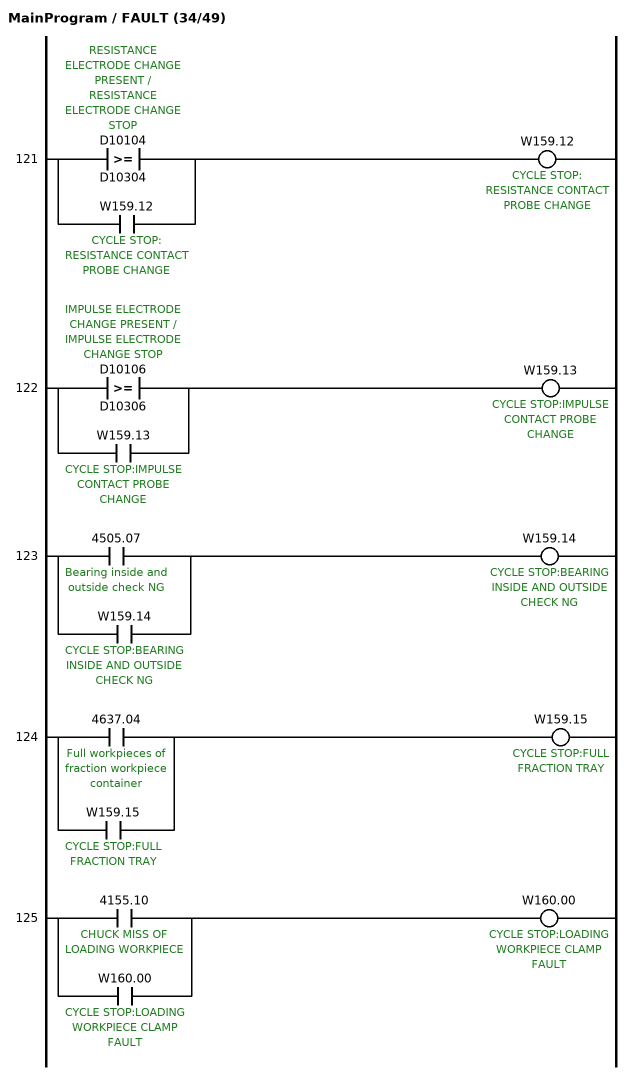
; [picture p96: MainProgram / FAULT, rungs 121-125]
; rung 121
LD>=L(326) D10104 D10304  ; RESISTANCE ELECTRODE CHANGE PRESENT, RESISTANCE ELECTRODE CHANGE STOP
OR W159.12  ; CYCLE STOP:RESISTANCE CONTACT PROBE CHANGE
OUT W159.12  ; CYCLE STOP:RESISTANCE CONTACT PROBE CHANGE
; rung 122
LD>=L(326) D10106 D10306  ; IMPULSE ELECTRODE CHANGE PRESENT, IMPULSE ELECTRODE CHANGE STOP
OR W159.13  ; CYCLE STOP:IMPULSE CONTACT PROBE CHANGE
OUT W159.13  ; CYCLE STOP:IMPULSE CONTACT PROBE CHANGE
; rung 123
LD 4505.07  ; Bearing inside and outside check NG
OR W159.14  ; CYCLE STOP:BEARING INSIDE AND OUTSIDE CHECK NG
OUT W159.14  ; CYCLE STOP:BEARING INSIDE AND OUTSIDE CHECK NG
; rung 124
LD 4637.04  ; Full workpieces of fraction workpiece container
OR W159.15  ; CYCLE STOP:FULL FRACTION TRAY
OUT W159.15  ; CYCLE STOP:FULL FRACTION TRAY
; rung 125
LD 4155.10  ; CHUCK MISS OF LOADING WORKPIECE
OR W160.00  ; CYCLE STOP:LOADING WORKPIECE CLAMP FAULT
OUT W160.00  ; CYCLE STOP:LOADING WORKPIECE CLAMP FAULT

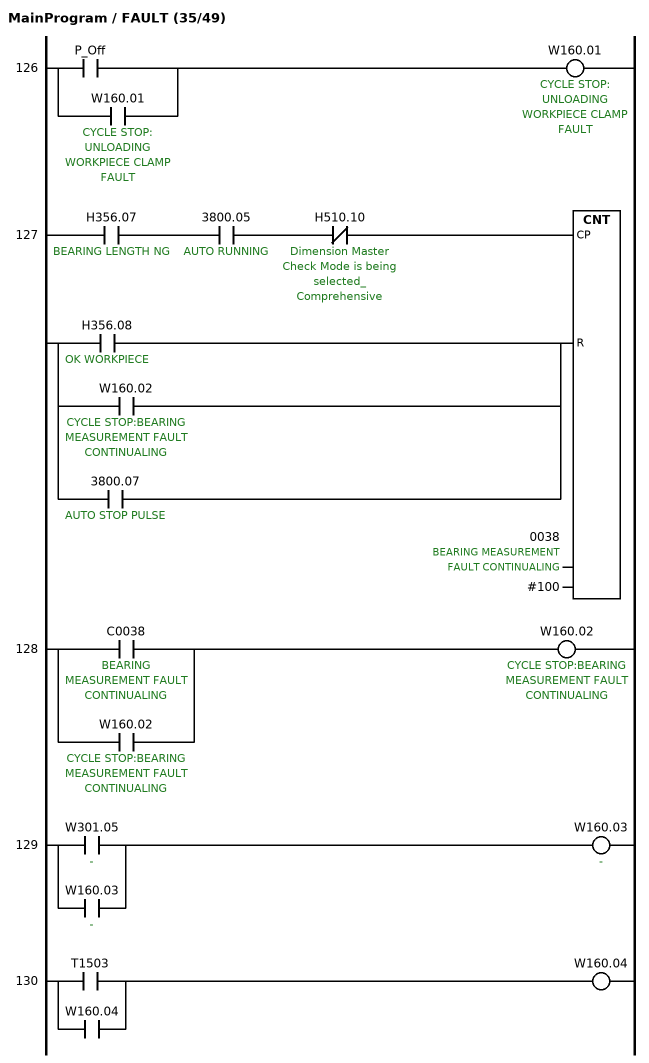
; rung 126
LD P_Off
OR W160.01  ; CYCLE STOP:UNLOADING WORKPIECE CLAMP FAULT
OUT W160.01  ; CYCLE STOP:UNLOADING WORKPIECE CLAMP FAULT
; rung 127
LD H356.07  ; BEARING LENGTH NG
AND 3800.05  ; AUTO RUNNING
ANDNOT H510.10  ; Dimension Master Check Mode is being selected_Comprehensive
LD H356.08  ; OK WORKPIECE
OR W160.02  ; CYCLE STOP:BEARING MEASUREMENT FAULT CONTINUALING
OR 3800.07  ; AUTO STOP PULSE
CNT 0038 #100  ; BEARING MEASUREMENT FAULT CONTINUALING
; rung 128
LD C0038  ; BEARING MEASUREMENT FAULT CONTINUALING
OR W160.02  ; CYCLE STOP:BEARING MEASUREMENT FAULT CONTINUALING
OUT W160.02  ; CYCLE STOP:BEARING MEASUREMENT FAULT CONTINUALING
; rung 129
LD W301.05  ; -
OR W160.03  ; -
OUT W160.03  ; -
; rung 130
LD T1503
OR W160.04
OUT W160.04

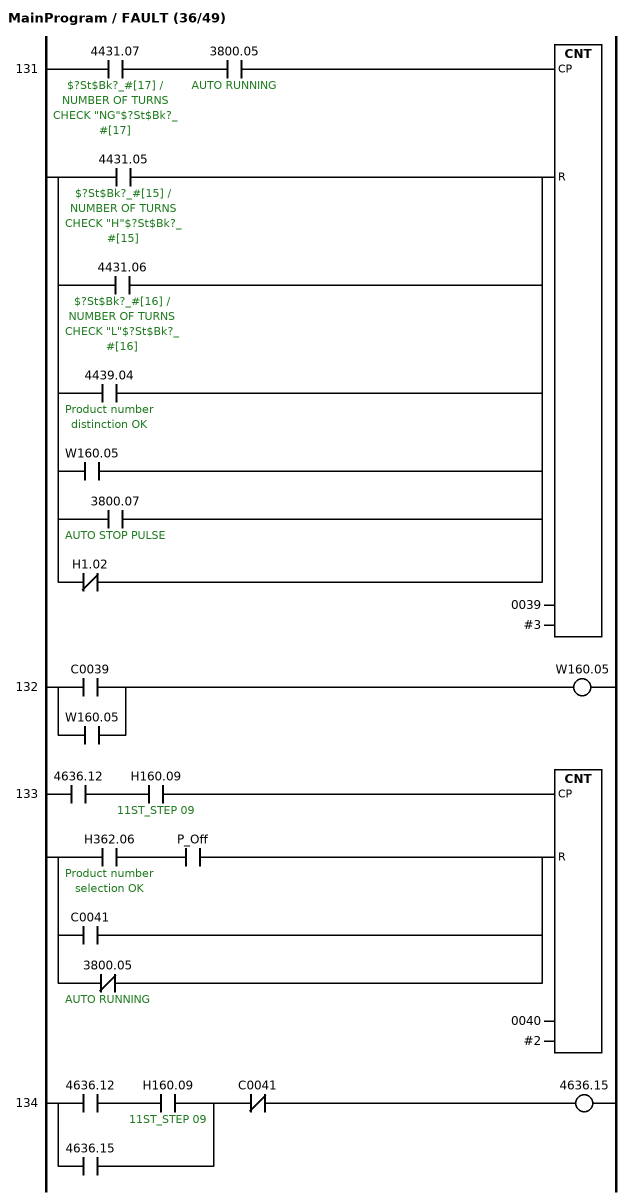
; rung 131
LD 4431.07  ; $?St$Bk?_#[17] / NUMBER OF TURNS CHECK "NG"$?St$Bk?_#[17]
AND 3800.05  ; AUTO RUNNING
LD 4431.05  ; $?St$Bk?_#[15] / NUMBER OF TURNS CHECK "H"$?St$Bk?_#[15]
OR 4431.06  ; $?St$Bk?_#[16] / NUMBER OF TURNS CHECK "L"$?St$Bk?_#[16]
OR 4439.04  ; Product number distinction OK
OR W160.05
OR 3800.07  ; AUTO STOP PULSE
ORNOT H1.02
CNT 0039 #3
; rung 132
LD C0039
OR W160.05
OUT W160.05
; rung 133
LD 4636.12
AND H160.09  ; 11ST_STEP 09
LD H362.06  ; Product number selection OK
AND P_Off
OR C0041
ORNOT 3800.05  ; AUTO RUNNING
CNT 0040 #2
; rung 134
LD 4636.12
AND H160.09  ; 11ST_STEP 09
OR 4636.15
ANDNOT C0041
OUT 4636.15

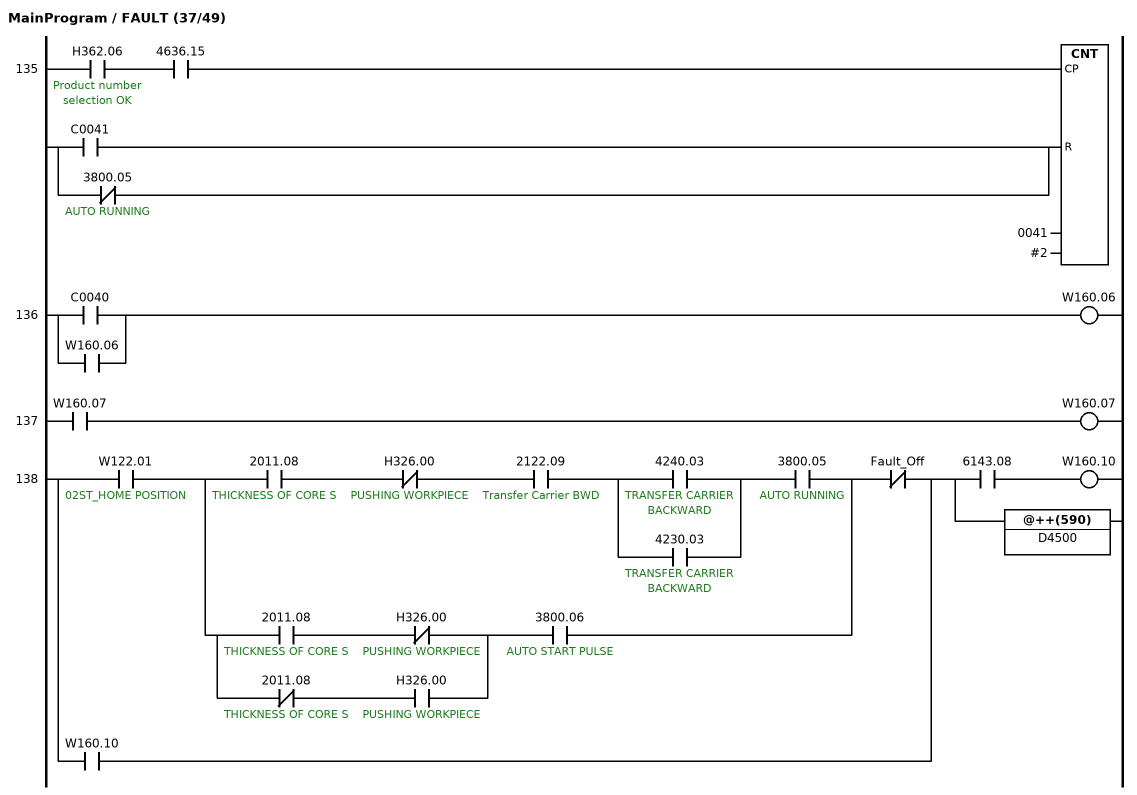
; rung 135
LD H362.06  ; Product number selection OK
AND 4636.15
LD C0041
ORNOT 3800.05  ; AUTO RUNNING
CNT 0041 #2
; rung 136
LD C0040
OR W160.06
OUT W160.06
; rung 137
LD W160.07
OUT W160.07
; rung 138
LD W122.01  ; 02ST_HOME POSITION
LD 2011.08  ; THICKNESS OF CORE S
ANDNOT H326.00  ; PUSHING WORKPIECE
AND 2122.09  ; Transfer Carrier BWD
LD 4240.03  ; TRANSFER CARRIER BACKWARD
OR 4230.03  ; TRANSFER CARRIER BACKWARD
ANDLD
AND 3800.05  ; AUTO RUNNING
LD 2011.08  ; THICKNESS OF CORE S
ANDNOT H326.00  ; PUSHING WORKPIECE
LDNOT 2011.08  ; THICKNESS OF CORE S
AND H326.00  ; PUSHING WORKPIECE
ORLD
AND 3800.06  ; AUTO START PULSE
ORLD
ANDLD
ANDNOT Fault_Off
OR W160.10
OUT TR0
AND 6143.08
OUT W160.10
LD TR0
@++(590) D4500

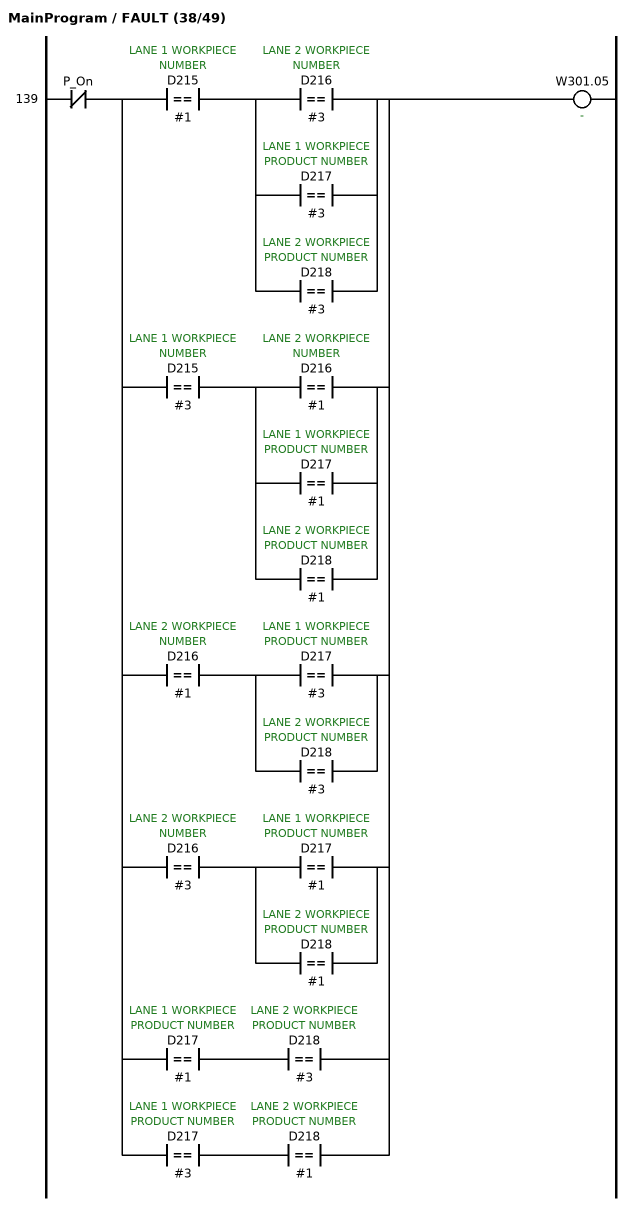
; rung 139
LDNOT P_On
LD=(300) D215 #1  ; LANE 1 WORKPIECE NUMBER
LD=(300) D216 #3  ; LANE 2 WORKPIECE NUMBER
OR=(300) D217 #3  ; LANE 1 WORKPIECE PRODUCT NUMBER
OR=(300) D218 #3  ; LANE 2 WORKPIECE PRODUCT NUMBER
ANDLD
LD=(300) D215 #3  ; LANE 1 WORKPIECE NUMBER
LD=(300) D216 #1  ; LANE 2 WORKPIECE NUMBER
OR=(300) D217 #1  ; LANE 1 WORKPIECE PRODUCT NUMBER
OR=(300) D218 #1  ; LANE 2 WORKPIECE PRODUCT NUMBER
ANDLD
ORLD
LD=(300) D216 #1  ; LANE 2 WORKPIECE NUMBER
LD=(300) D217 #3  ; LANE 1 WORKPIECE PRODUCT NUMBER
OR=(300) D218 #3  ; LANE 2 WORKPIECE PRODUCT NUMBER
ANDLD
ORLD
LD=(300) D216 #3  ; LANE 2 WORKPIECE NUMBER
LD=(300) D217 #1  ; LANE 1 WORKPIECE PRODUCT NUMBER
OR=(300) D218 #1  ; LANE 2 WORKPIECE PRODUCT NUMBER
ANDLD
ORLD
LD=(300) D217 #1  ; LANE 1 WORKPIECE PRODUCT NUMBER
AND=(300) D218 #3  ; LANE 2 WORKPIECE PRODUCT NUMBER
ORLD
LD=(300) D217 #3  ; LANE 1 WORKPIECE PRODUCT NUMBER
AND=(300) D218 #1  ; LANE 2 WORKPIECE PRODUCT NUMBER
ORLD
ANDLD
OUT W301.05  ; -

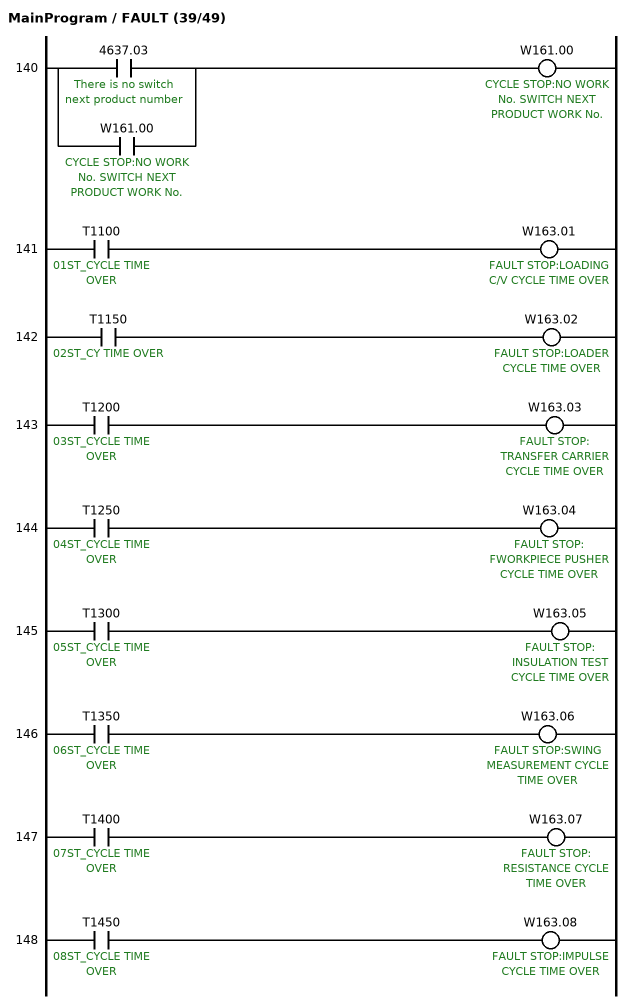
; rung 140
LD 4637.03  ; There is no switch next product number
OR W161.00  ; CYCLE STOP:NO WORK No. SWITCH NEXT PRODUCT WORK No.
OUT W161.00  ; CYCLE STOP:NO WORK No. SWITCH NEXT PRODUCT WORK No.
; rung 141
LD T1100  ; 01ST_CYCLE TIME OVER
OUT W163.01  ; FAULT STOP:LOADING C/V CYCLE TIME OVER
; rung 142
LD T1150  ; 02ST_CY TIME OVER
OUT W163.02  ; FAULT STOP:LOADER CYCLE TIME OVER
; rung 143
LD T1200  ; 03ST_CYCLE TIME OVER
OUT W163.03  ; FAULT STOP:TRANSFER CARRIER CYCLE TIME OVER
; rung 144
LD T1250  ; 04ST_CYCLE TIME OVER
OUT W163.04  ; FAULT STOP:FWORKPIECE PUSHER CYCLE TIME OVER
; rung 145
LD T1300  ; 05ST_CYCLE TIME OVER
OUT W163.05  ; FAULT STOP:INSULATION TEST CYCLE TIME OVER
; rung 146
LD T1350  ; 06ST_CYCLE TIME OVER
OUT W163.06  ; FAULT STOP:SWING MEASUREMENT CYCLE TIME OVER
; rung 147
LD T1400  ; 07ST_CYCLE TIME OVER
OUT W163.07  ; FAULT STOP:RESISTANCE CYCLE TIME OVER
; rung 148
LD T1450  ; 08ST_CYCLE TIME OVER
OUT W163.08  ; FAULT STOP:IMPULSE CYCLE TIME OVER

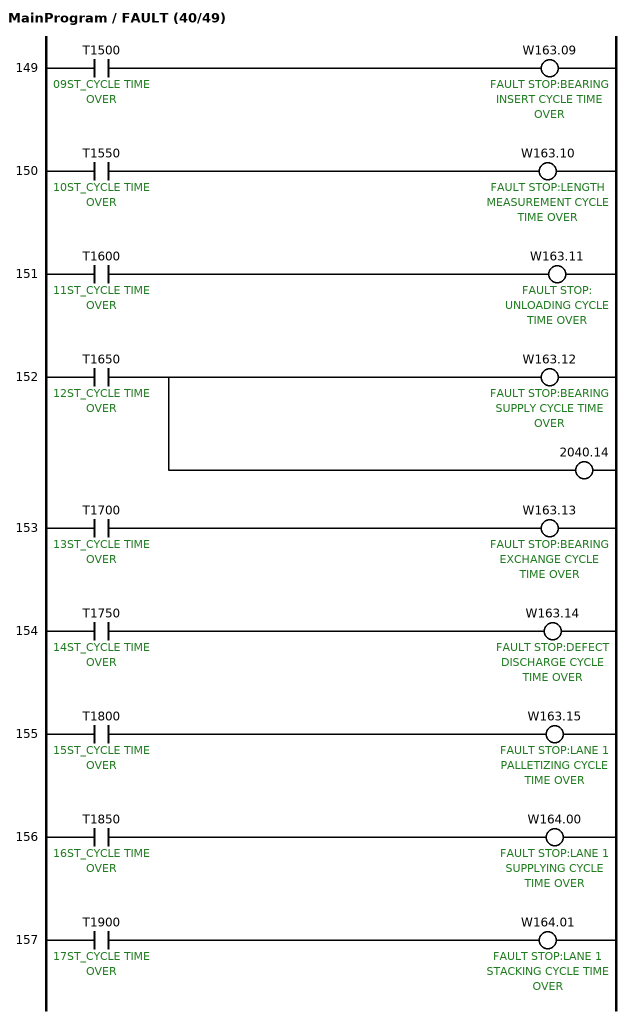
; rung 149
LD T1500  ; 09ST_CYCLE TIME OVER
OUT W163.09  ; FAULT STOP:BEARING INSERT CYCLE TIME OVER
; rung 150
LD T1550  ; 10ST_CYCLE TIME OVER
OUT W163.10  ; FAULT STOP:LENGTH MEASUREMENT CYCLE TIME OVER
; rung 151
LD T1600  ; 11ST_CYCLE TIME OVER
OUT W163.11  ; FAULT STOP:UNLOADING CYCLE TIME OVER
; rung 152
LD T1650  ; 12ST_CYCLE TIME OVER
OUT W163.12  ; FAULT STOP:BEARING SUPPLY CYCLE TIME OVER
OUT 2040.14
; rung 153
LD T1700  ; 13ST_CYCLE TIME OVER
OUT W163.13  ; FAULT STOP:BEARING EXCHANGE CYCLE TIME OVER
; rung 154
LD T1750  ; 14ST_CYCLE TIME OVER
OUT W163.14  ; FAULT STOP:DEFECT DISCHARGE CYCLE TIME OVER
; rung 155
LD T1800  ; 15ST_CYCLE TIME OVER
OUT W163.15  ; FAULT STOP:LANE 1 PALLETIZING CYCLE TIME OVER
; rung 156
LD T1850  ; 16ST_CYCLE TIME OVER
OUT W164.00  ; FAULT STOP:LANE 1 SUPPLYING CYCLE TIME OVER
; rung 157
LD T1900  ; 17ST_CYCLE TIME OVER
OUT W164.01  ; FAULT STOP:LANE 1 STACKING CYCLE TIME OVER

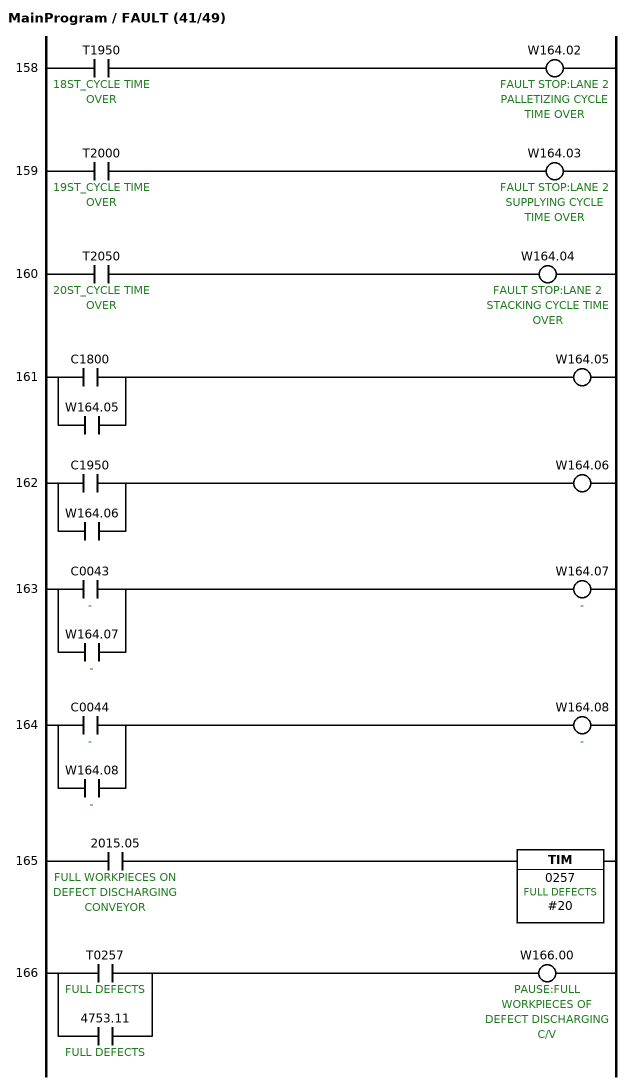
; rung 158
LD T1950  ; 18ST_CYCLE TIME OVER
OUT W164.02  ; FAULT STOP:LANE 2 PALLETIZING CYCLE TIME OVER
; rung 159
LD T2000  ; 19ST_CYCLE TIME OVER
OUT W164.03  ; FAULT STOP:LANE 2 SUPPLYING CYCLE TIME OVER
; rung 160
LD T2050  ; 20ST_CYCLE TIME OVER
OUT W164.04  ; FAULT STOP:LANE 2 STACKING CYCLE TIME OVER
; rung 161
LD C1800
OR W164.05
OUT W164.05
; rung 162
LD C1950
OR W164.06
OUT W164.06
; rung 163
LD C0043  ; -
OR W164.07  ; -
OUT W164.07  ; -
; rung 164
LD C0044  ; -
OR W164.08  ; -
OUT W164.08  ; -
; rung 165
LD 2015.05  ; FULL WORKPIECES ON DEFECT DISCHARGING CONVEYOR
TIM 0257 #20  ; FULL DEFECTS
; rung 166
LD T0257  ; FULL DEFECTS
OR 4753.11  ; FULL DEFECTS
OUT W166.00  ; PAUSE:FULL WORKPIECES OF DEFECT DISCHARGING C/V

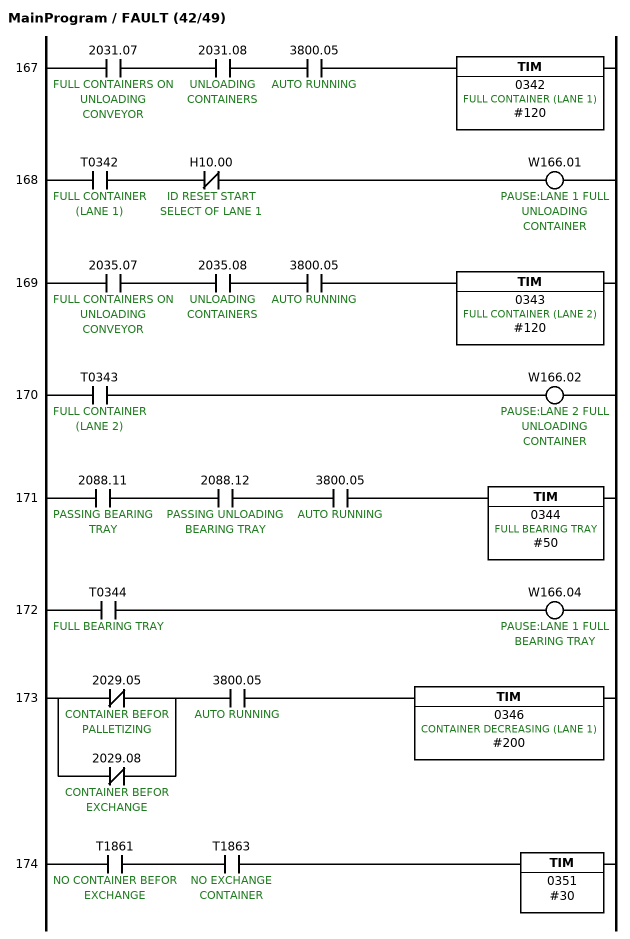
; rung 167
LD 2031.07  ; FULL CONTAINERS ON UNLOADING CONVEYOR
AND 2031.08  ; UNLOADING CONTAINERS
AND 3800.05  ; AUTO RUNNING
TIM 0342 #120  ; FULL CONTAINER (LANE 1)
; rung 168
LD T0342  ; FULL CONTAINER (LANE 1)
ANDNOT H10.00  ; ID RESET START SELECT OF LANE 1
OUT W166.01  ; PAUSE:LANE 1 FULL UNLOADING CONTAINER
; rung 169
LD 2035.07  ; FULL CONTAINERS ON UNLOADING CONVEYOR
AND 2035.08  ; UNLOADING CONTAINERS
AND 3800.05  ; AUTO RUNNING
TIM 0343 #120  ; FULL CONTAINER (LANE 2)
; rung 170
LD T0343  ; FULL CONTAINER (LANE 2)
OUT W166.02  ; PAUSE:LANE 2 FULL UNLOADING CONTAINER
; rung 171
LD 2088.11  ; PASSING BEARING TRAY
AND 2088.12  ; PASSING UNLOADING BEARING TRAY
AND 3800.05  ; AUTO RUNNING
TIM 0344 #50  ; FULL BEARING TRAY
; rung 172
LD T0344  ; FULL BEARING TRAY
OUT W166.04  ; PAUSE:LANE 1 FULL BEARING TRAY
; rung 173
LDNOT 2029.05  ; CONTAINER BEFOR PALLETIZING
ORNOT 2029.08  ; CONTAINER BEFOR EXCHANGE
AND 3800.05  ; AUTO RUNNING
TIM 0346 #200  ; CONTAINER DECREASING (LANE 1)
; rung 174
LD T1861  ; NO CONTAINER BEFOR EXCHANGE
AND T1863  ; NO EXCHANGE CONTAINER
TIM 0351 #30

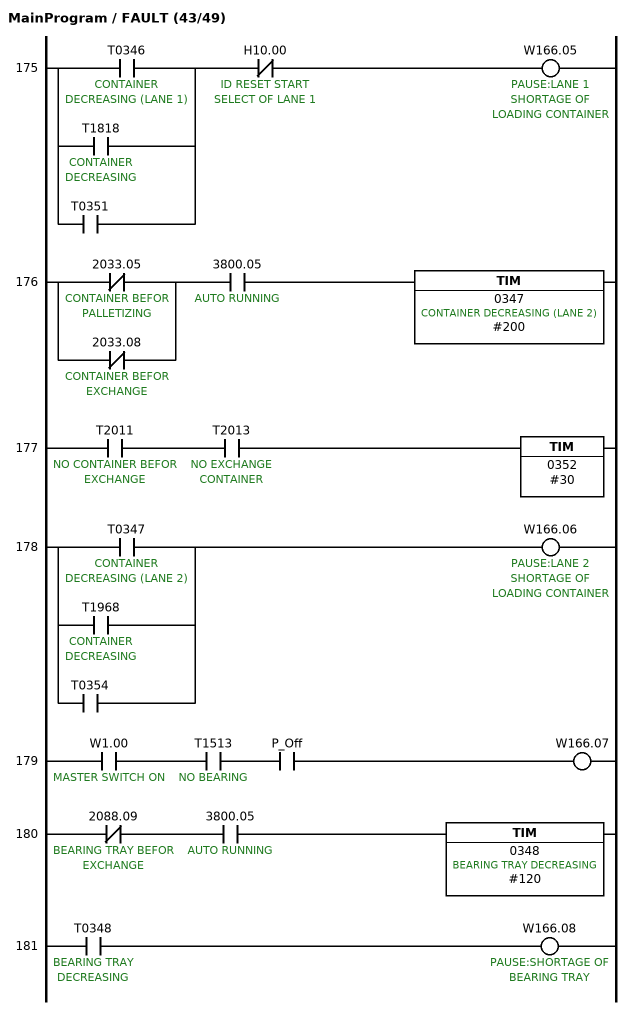
; rung 175
LD T0346  ; CONTAINER DECREASING (LANE 1)
OR T1818  ; CONTAINER DECREASING
OR T0351
ANDNOT H10.00  ; ID RESET START SELECT OF LANE 1
OUT W166.05  ; PAUSE:LANE 1 SHORTAGE OF LOADING CONTAINER
; rung 176
LDNOT 2033.05  ; CONTAINER BEFOR PALLETIZING
ORNOT 2033.08  ; CONTAINER BEFOR EXCHANGE
AND 3800.05  ; AUTO RUNNING
TIM 0347 #200  ; CONTAINER DECREASING (LANE 2)
; rung 177
LD T2011  ; NO CONTAINER BEFOR EXCHANGE
AND T2013  ; NO EXCHANGE CONTAINER
TIM 0352 #30
; rung 178
LD T0347  ; CONTAINER DECREASING (LANE 2)
OR T1968  ; CONTAINER DECREASING
OR T0354
OUT W166.06  ; PAUSE:LANE 2 SHORTAGE OF LOADING CONTAINER
; rung 179
LD W1.00  ; MASTER SWITCH ON
AND T1513  ; NO BEARING
AND P_Off
OUT W166.07
; rung 180
LDNOT 2088.09  ; BEARING TRAY BEFOR EXCHANGE
AND 3800.05  ; AUTO RUNNING
TIM 0348 #120  ; BEARING TRAY DECREASING
; rung 181
LD T0348  ; BEARING TRAY DECREASING
OUT W166.08  ; PAUSE:SHORTAGE OF BEARING TRAY

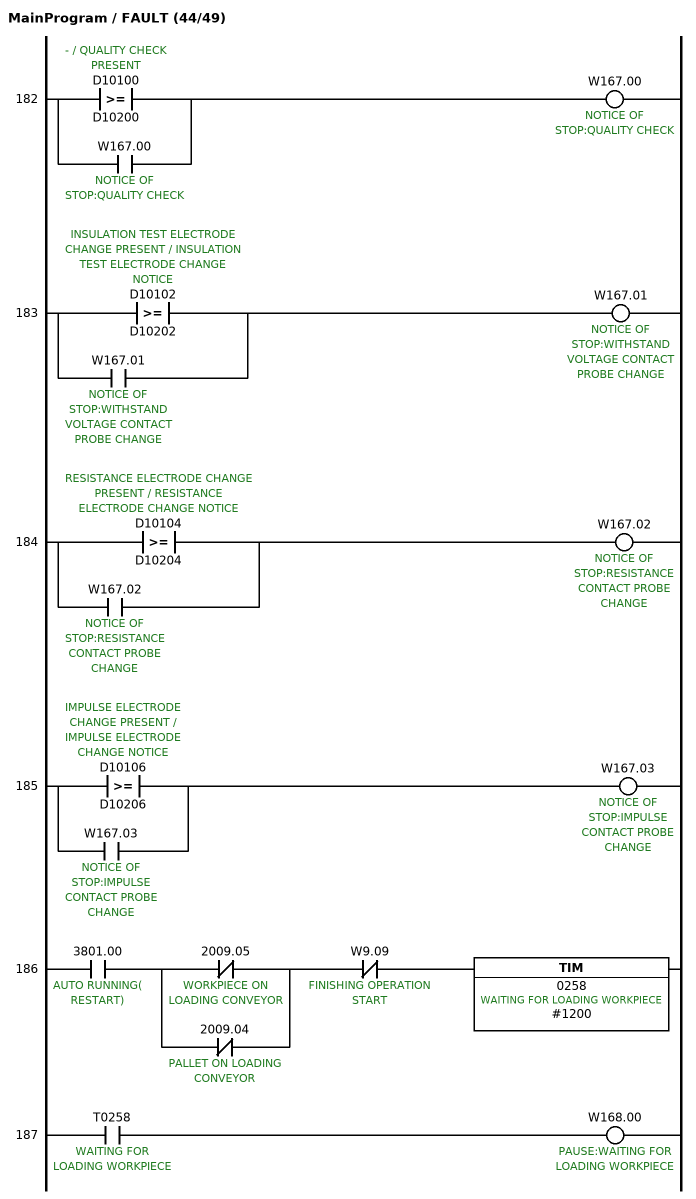
; rung 182
LD>=L(326) D10100 D10200  ; -, QUALITY CHECK PRESENT
OR W167.00  ; NOTICE OF STOP:QUALITY CHECK
OUT W167.00  ; NOTICE OF STOP:QUALITY CHECK
; rung 183
LD>=L(326) D10102 D10202  ; INSULATION TEST ELECTRODE CHANGE PRESENT, INSULATION TEST ELECTRODE CHANGE NOTICE
OR W167.01  ; NOTICE OF STOP:WITHSTAND VOLTAGE CONTACT PROBE CHANGE
OUT W167.01  ; NOTICE OF STOP:WITHSTAND VOLTAGE CONTACT PROBE CHANGE
; rung 184
LD>=L(326) D10104 D10204  ; RESISTANCE ELECTRODE CHANGE PRESENT, RESISTANCE ELECTRODE CHANGE NOTICE
OR W167.02  ; NOTICE OF STOP:RESISTANCE CONTACT PROBE CHANGE
OUT W167.02  ; NOTICE OF STOP:RESISTANCE CONTACT PROBE CHANGE
; rung 185
LD>=L(326) D10106 D10206  ; IMPULSE ELECTRODE CHANGE PRESENT, IMPULSE ELECTRODE CHANGE NOTICE
OR W167.03  ; NOTICE OF STOP:IMPULSE CONTACT PROBE CHANGE
OUT W167.03  ; NOTICE OF STOP:IMPULSE CONTACT PROBE CHANGE
; rung 186
LD 3801.00  ; AUTO RUNNING(RESTART)
LDNOT 2009.05  ; WORKPIECE ON LOADING CONVEYOR
ORNOT 2009.04  ; PALLET ON LOADING CONVEYOR
ANDLD
ANDNOT W9.09  ; FINISHING OPERATION START
TIM 0258 #1200  ; WAITING FOR LOADING WORKPIECE
; rung 187
LD T0258  ; WAITING FOR LOADING WORKPIECE
OUT W168.00  ; PAUSE:WAITING FOR LOADING WORKPIECE

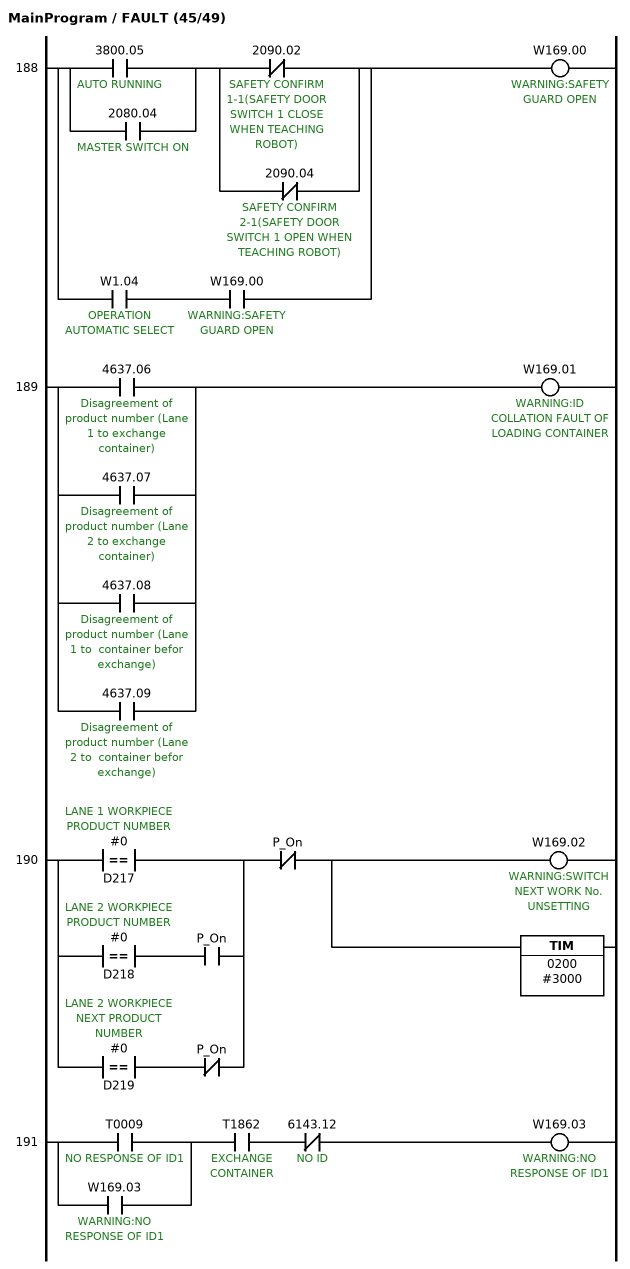
; rung 188
LD 3800.05  ; AUTO RUNNING
OR 2080.04  ; MASTER SWITCH ON
LDNOT 2090.02  ; SAFETY CONFIRM 1-1(SAFETY DOOR SWITCH 1 CLOSE WHEN TEACHING ROBOT)
ORNOT 2090.04  ; SAFETY CONFIRM 2-1(SAFETY DOOR SWITCH 1 OPEN WHEN TEACHING ROBOT)
ANDLD
LD W1.04  ; OPERATION AUTOMATIC SELECT
AND W169.00  ; WARNING:SAFETY GUARD OPEN
ORLD
OUT W169.00  ; WARNING:SAFETY GUARD OPEN
; rung 189
LD 4637.06  ; Disagreement of product number (Lane 1 to exchange container)
OR 4637.07  ; Disagreement of product number (Lane 2 to exchange container)
OR 4637.08  ; Disagreement of product number (Lane 1 to  container befor exchange)
OR 4637.09  ; Disagreement of product number (Lane 2 to  container befor exchange)
OUT W169.01  ; WARNING:ID COLLATION FAULT OF LOADING CONTAINER
; rung 190
LD=(300) #0 D217  ; LANE 1 WORKPIECE PRODUCT NUMBER
LD=(300) #0 D218  ; LANE 2 WORKPIECE PRODUCT NUMBER
AND P_On
ORLD
LD=(300) #0 D219  ; LANE 2 WORKPIECE NEXT PRODUCT NUMBER
ANDNOT P_On
ORLD
ANDNOT P_On
OUT W169.02  ; WARNING:SWITCH NEXT WORK No. UNSETTING
TIM 0200 #3000
; rung 191
LD T0009  ; NO RESPONSE OF ID1
OR W169.03  ; WARNING:NO RESPONSE OF ID1
AND T1862  ; EXCHANGE CONTAINER
ANDNOT 6143.12  ; NO ID
OUT W169.03  ; WARNING:NO RESPONSE OF ID1

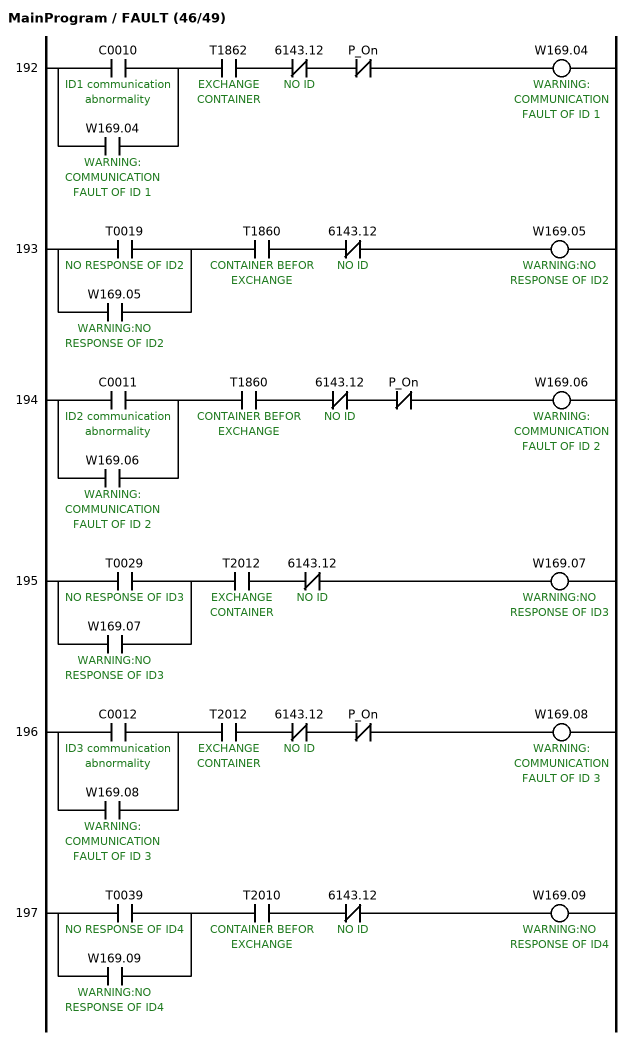
; rung 192
LD C0010  ; ID1 communication abnormality
OR W169.04  ; WARNING:COMMUNICATION FAULT OF ID 1
AND T1862  ; EXCHANGE CONTAINER
ANDNOT 6143.12  ; NO ID
ANDNOT P_On
OUT W169.04  ; WARNING:COMMUNICATION FAULT OF ID 1
; rung 193
LD T0019  ; NO RESPONSE OF ID2
OR W169.05  ; WARNING:NO RESPONSE OF ID2
AND T1860  ; CONTAINER BEFOR EXCHANGE
ANDNOT 6143.12  ; NO ID
OUT W169.05  ; WARNING:NO RESPONSE OF ID2
; rung 194
LD C0011  ; ID2 communication abnormality
OR W169.06  ; WARNING:COMMUNICATION FAULT OF ID 2
AND T1860  ; CONTAINER BEFOR EXCHANGE
ANDNOT 6143.12  ; NO ID
ANDNOT P_On
OUT W169.06  ; WARNING:COMMUNICATION FAULT OF ID 2
; rung 195
LD T0029  ; NO RESPONSE OF ID3
OR W169.07  ; WARNING:NO RESPONSE OF ID3
AND T2012  ; EXCHANGE CONTAINER
ANDNOT 6143.12  ; NO ID
OUT W169.07  ; WARNING:NO RESPONSE OF ID3
; rung 196
LD C0012  ; ID3 communication abnormality
OR W169.08  ; WARNING:COMMUNICATION FAULT OF ID 3
AND T2012  ; EXCHANGE CONTAINER
ANDNOT 6143.12  ; NO ID
ANDNOT P_On
OUT W169.08  ; WARNING:COMMUNICATION FAULT OF ID 3
; rung 197
LD T0039  ; NO RESPONSE OF ID4
OR W169.09  ; WARNING:NO RESPONSE OF ID4
AND T2010  ; CONTAINER BEFOR EXCHANGE
ANDNOT 6143.12  ; NO ID
OUT W169.09  ; WARNING:NO RESPONSE OF ID4

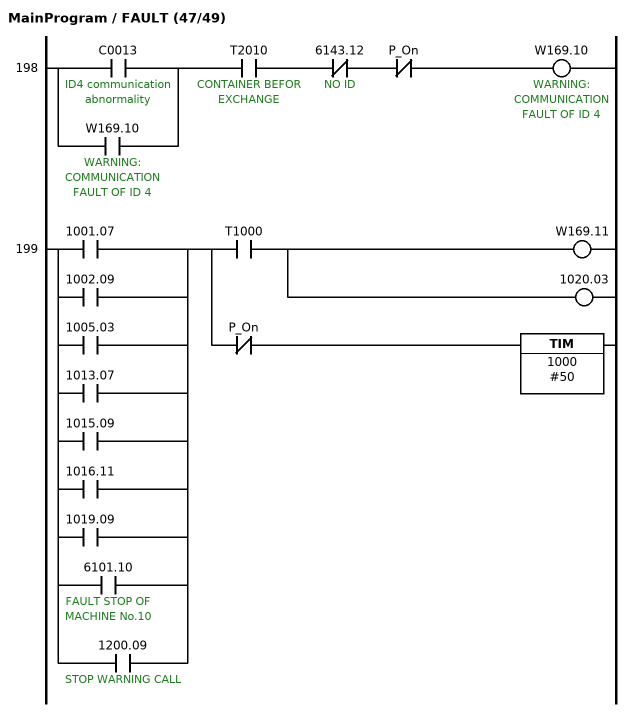
; rung 198
LD C0013  ; ID4 communication abnormality
OR W169.10  ; WARNING:COMMUNICATION FAULT OF ID 4
AND T2010  ; CONTAINER BEFOR EXCHANGE
ANDNOT 6143.12  ; NO ID
ANDNOT P_On
OUT W169.10  ; WARNING:COMMUNICATION FAULT OF ID 4
; rung 199
LD 1001.07
OR 1002.09
OR 1005.03
OR 1013.07
OR 1015.09
OR 1016.11
OR 1019.09
OR 6101.10  ; FAULT STOP OF MACHINE No.10
OR 1200.09  ; STOP WARNING CALL
OUT TR0
AND T1000
OUT W169.11
OUT 1020.03
LD TR0
ANDNOT P_On
TIM 1000 #50

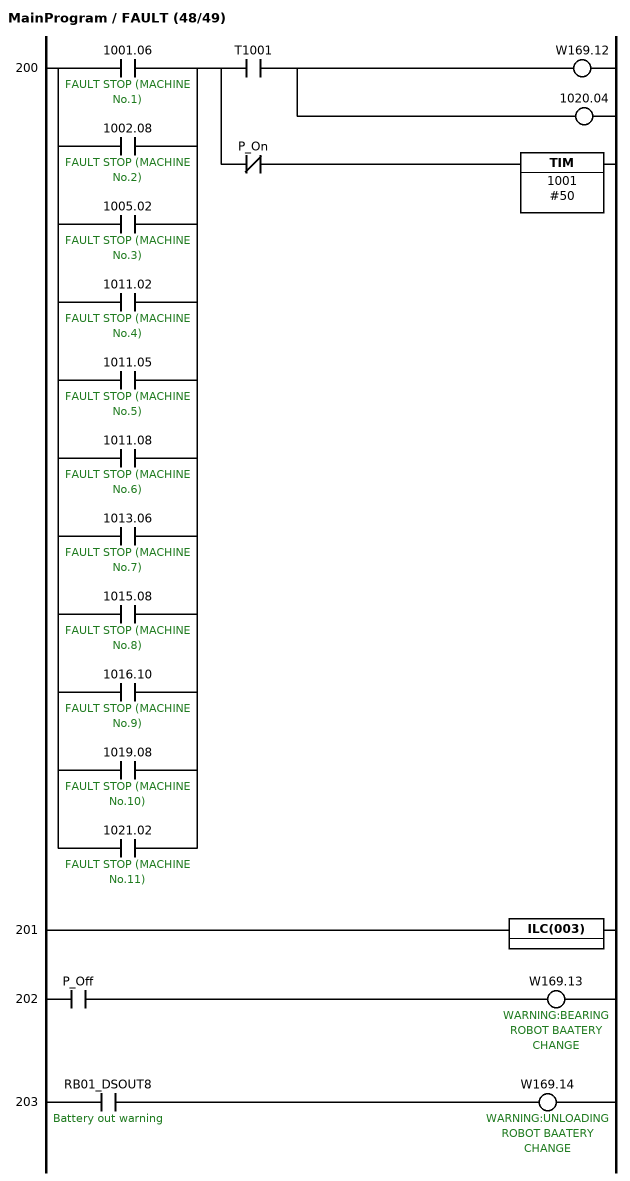
; rung 200
LD 1001.06  ; FAULT STOP (MACHINE No.1)
OR 1002.08  ; FAULT STOP (MACHINE No.2)
OR 1005.02  ; FAULT STOP (MACHINE No.3)
OR 1011.02  ; FAULT STOP (MACHINE No.4)
OR 1011.05  ; FAULT STOP (MACHINE No.5)
OR 1011.08  ; FAULT STOP (MACHINE No.6)
OR 1013.06  ; FAULT STOP (MACHINE No.7)
OR 1015.08  ; FAULT STOP (MACHINE No.8)
OR 1016.10  ; FAULT STOP (MACHINE No.9)
OR 1019.08  ; FAULT STOP (MACHINE No.10)
OR 1021.02  ; FAULT STOP (MACHINE No.11)
OUT TR0
AND T1001
OUT W169.12
OUT 1020.04
LD TR0
ANDNOT P_On
TIM 1001 #50
; rung 201
ILC(003)
; rung 202
LD P_Off
OUT W169.13  ; WARNING:BEARING ROBOT BAATERY CHANGE
; rung 203
LD RB01_DSOUT8  ; Battery out warning
OUT W169.14  ; WARNING:UNLOADING ROBOT BAATERY CHANGE

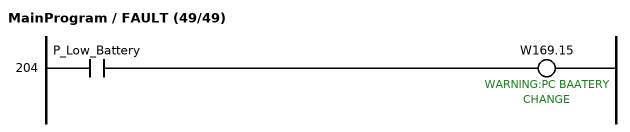
; rung 204
LD P_Low_Battery
OUT W169.15  ; WARNING:PC BAATERY CHANGE

### Section UNIT_FAULT_DISPLAY

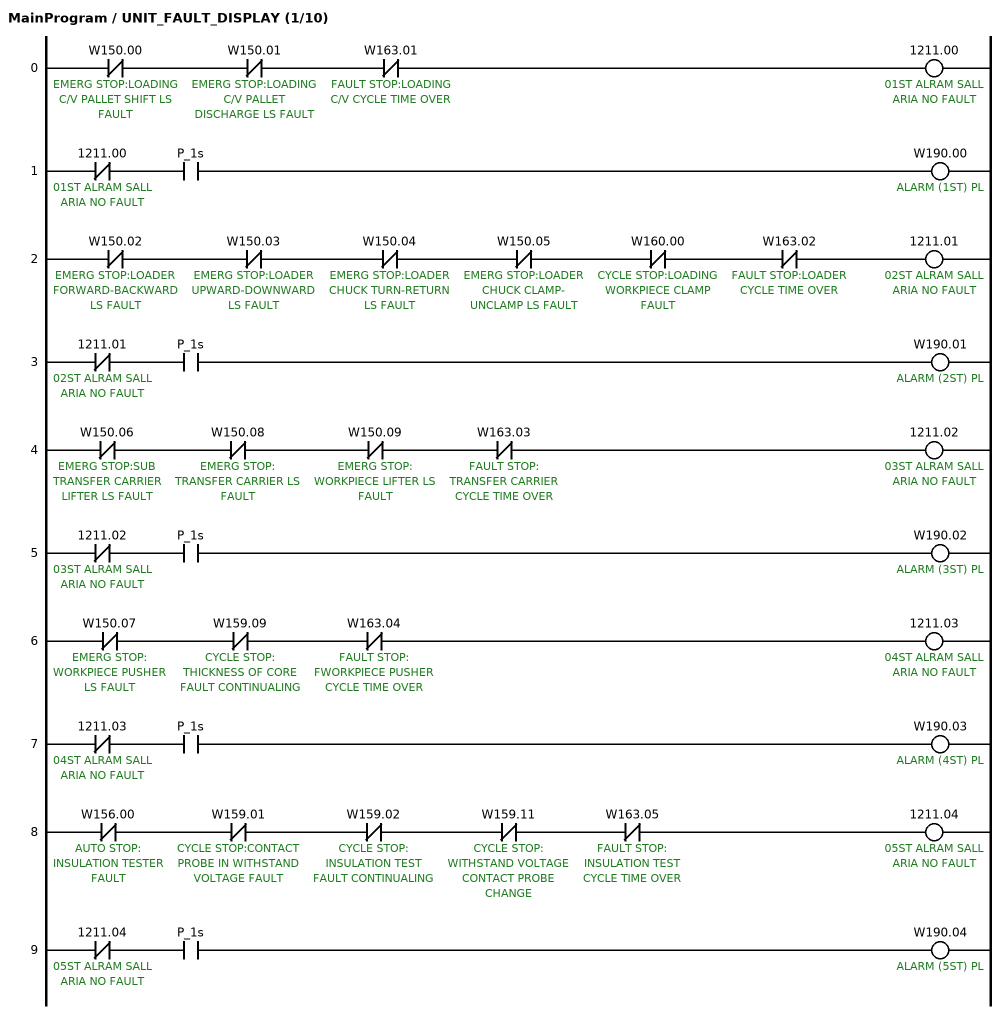
; rung 0
LDNOT W150.00  ; EMERG STOP:LOADING C/V PALLET SHIFT LS FAULT
ANDNOT W150.01  ; EMERG STOP:LOADING C/V PALLET DISCHARGE LS FAULT
ANDNOT W163.01  ; FAULT STOP:LOADING C/V CYCLE TIME OVER
OUT 1211.00  ; 01ST ALRAM SALL ARIA NO FAULT
; rung 1
LDNOT 1211.00  ; 01ST ALRAM SALL ARIA NO FAULT
AND P_1s
OUT W190.00  ; ALARM (1ST) PL
; rung 2
LDNOT W150.02  ; EMERG STOP:LOADER FORWARD-BACKWARD LS FAULT
ANDNOT W150.03  ; EMERG STOP:LOADER UPWARD-DOWNWARD LS FAULT
ANDNOT W150.04  ; EMERG STOP:LOADER CHUCK TURN-RETURN LS FAULT
ANDNOT W150.05  ; EMERG STOP:LOADER CHUCK CLAMP-UNCLAMP LS FAULT
ANDNOT W160.00  ; CYCLE STOP:LOADING WORKPIECE CLAMP FAULT
ANDNOT W163.02  ; FAULT STOP:LOADER CYCLE TIME OVER
OUT 1211.01  ; 02ST ALRAM SALL ARIA NO FAULT
; rung 3
LDNOT 1211.01  ; 02ST ALRAM SALL ARIA NO FAULT
AND P_1s
OUT W190.01  ; ALARM (2ST) PL
; rung 4
LDNOT W150.06  ; EMERG STOP:SUB TRANSFER CARRIER LIFTER LS FAULT
ANDNOT W150.08  ; EMERG STOP:TRANSFER CARRIER LS FAULT
ANDNOT W150.09  ; EMERG STOP:WORKPIECE LIFTER LS FAULT
ANDNOT W163.03  ; FAULT STOP:TRANSFER CARRIER CYCLE TIME OVER
OUT 1211.02  ; 03ST ALRAM SALL ARIA NO FAULT
; rung 5
LDNOT 1211.02  ; 03ST ALRAM SALL ARIA NO FAULT
AND P_1s
OUT W190.02  ; ALARM (3ST) PL
; rung 6
LDNOT W150.07  ; EMERG STOP:WORKPIECE PUSHER LS FAULT
ANDNOT W159.09  ; CYCLE STOP:THICKNESS OF CORE FAULT CONTINUALING
ANDNOT W163.04  ; FAULT STOP:FWORKPIECE PUSHER CYCLE TIME OVER
OUT 1211.03  ; 04ST ALRAM SALL ARIA NO FAULT
; rung 7
LDNOT 1211.03  ; 04ST ALRAM SALL ARIA NO FAULT
AND P_1s
OUT W190.03  ; ALARM (4ST) PL
; rung 8
LDNOT W156.00  ; AUTO STOP:INSULATION TESTER FAULT
ANDNOT W159.01  ; CYCLE STOP:CONTACT PROBE IN WITHSTAND VOLTAGE FAULT
ANDNOT W159.02  ; CYCLE STOP:INSULATION TEST FAULT CONTINUALING
ANDNOT W159.11  ; CYCLE STOP:WITHSTAND VOLTAGE CONTACT PROBE CHANGE
ANDNOT W163.05  ; FAULT STOP:INSULATION TEST CYCLE TIME OVER
OUT 1211.04  ; 05ST ALRAM SALL ARIA NO FAULT
; rung 9
LDNOT 1211.04  ; 05ST ALRAM SALL ARIA NO FAULT
AND P_1s
OUT W190.04  ; ALARM (5ST) PL

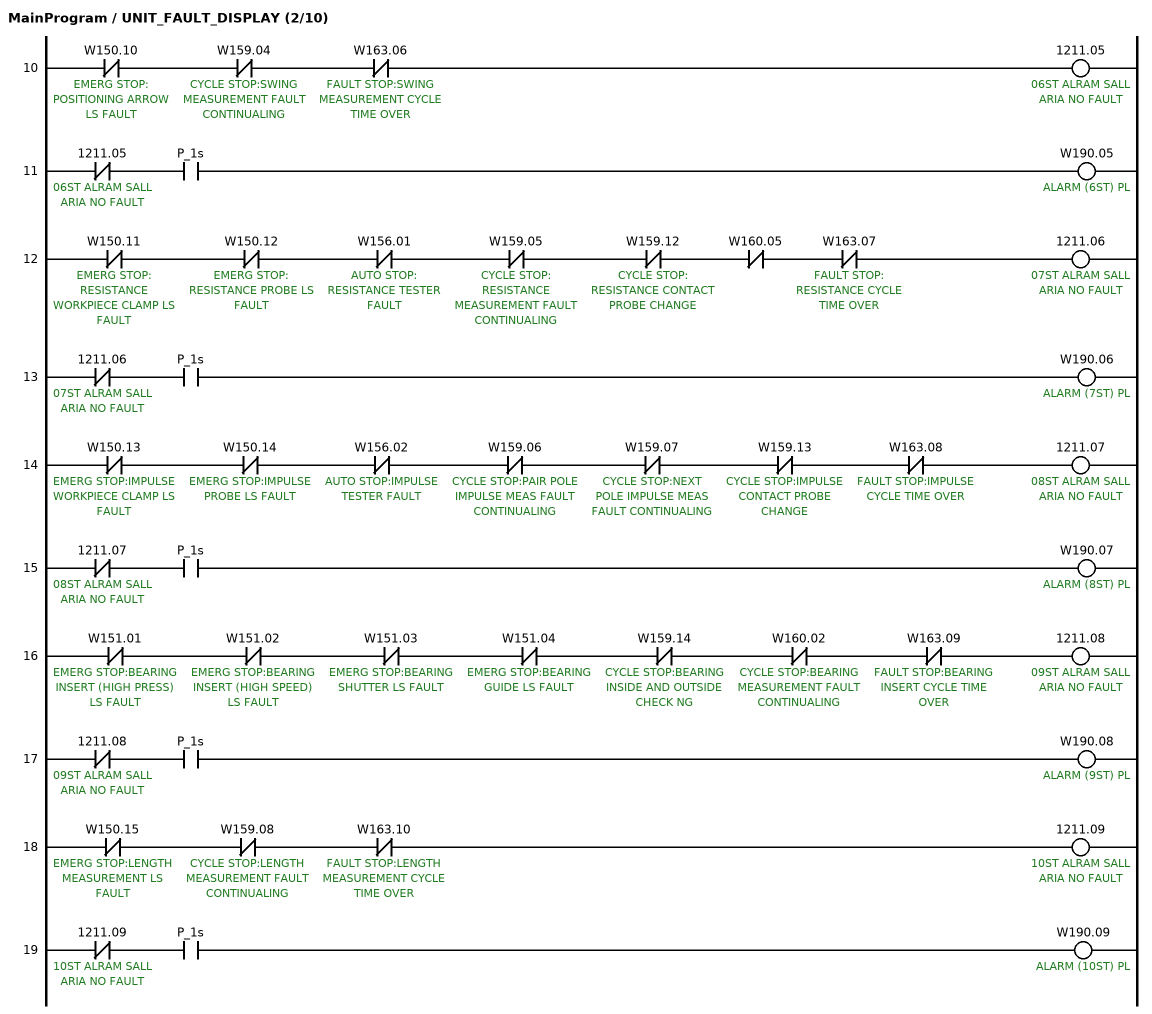
; rung 10
LDNOT W150.10  ; EMERG STOP:POSITIONING ARROW LS FAULT
ANDNOT W159.04  ; CYCLE STOP:SWING MEASUREMENT FAULT CONTINUALING
ANDNOT W163.06  ; FAULT STOP:SWING MEASUREMENT CYCLE TIME OVER
OUT 1211.05  ; 06ST ALRAM SALL ARIA NO FAULT
; rung 11
LDNOT 1211.05  ; 06ST ALRAM SALL ARIA NO FAULT
AND P_1s
OUT W190.05  ; ALARM (6ST) PL
; rung 12
LDNOT W150.11  ; EMERG STOP:RESISTANCE WORKPIECE CLAMP LS FAULT
ANDNOT W150.12  ; EMERG STOP:RESISTANCE PROBE LS FAULT
ANDNOT W156.01  ; AUTO STOP:RESISTANCE TESTER FAULT
ANDNOT W159.05  ; CYCLE STOP:RESISTANCE MEASUREMENT FAULT CONTINUALING
ANDNOT W159.12  ; CYCLE STOP:RESISTANCE CONTACT PROBE CHANGE
ANDNOT W160.05
ANDNOT W163.07  ; FAULT STOP:RESISTANCE CYCLE TIME OVER
OUT 1211.06  ; 07ST ALRAM SALL ARIA NO FAULT
; rung 13
LDNOT 1211.06  ; 07ST ALRAM SALL ARIA NO FAULT
AND P_1s
OUT W190.06  ; ALARM (7ST) PL
; rung 14
LDNOT W150.13  ; EMERG STOP:IMPULSE WORKPIECE CLAMP LS FAULT
ANDNOT W150.14  ; EMERG STOP:IMPULSE PROBE LS FAULT
ANDNOT W156.02  ; AUTO STOP:IMPULSE TESTER FAULT
ANDNOT W159.06  ; CYCLE STOP:PAIR POLE IMPULSE MEAS FAULT CONTINUALING
ANDNOT W159.07  ; CYCLE STOP:NEXT POLE IMPULSE MEAS FAULT CONTINUALING
ANDNOT W159.13  ; CYCLE STOP:IMPULSE CONTACT PROBE CHANGE
ANDNOT W163.08  ; FAULT STOP:IMPULSE CYCLE TIME OVER
OUT 1211.07  ; 08ST ALRAM SALL ARIA NO FAULT
; rung 15
LDNOT 1211.07  ; 08ST ALRAM SALL ARIA NO FAULT
AND P_1s
OUT W190.07  ; ALARM (8ST) PL
; rung 16
LDNOT W151.01  ; EMERG STOP:BEARING INSERT (HIGH PRESS) LS FAULT
ANDNOT W151.02  ; EMERG STOP:BEARING INSERT (HIGH SPEED) LS FAULT
ANDNOT W151.03  ; EMERG STOP:BEARING SHUTTER LS FAULT
ANDNOT W151.04  ; EMERG STOP:BEARING GUIDE LS FAULT
ANDNOT W159.14  ; CYCLE STOP:BEARING INSIDE AND OUTSIDE CHECK NG
ANDNOT W160.02  ; CYCLE STOP:BEARING MEASUREMENT FAULT CONTINUALING
ANDNOT W163.09  ; FAULT STOP:BEARING INSERT CYCLE TIME OVER
OUT 1211.08  ; 09ST ALRAM SALL ARIA NO FAULT
; rung 17
LDNOT 1211.08  ; 09ST ALRAM SALL ARIA NO FAULT
AND P_1s
OUT W190.08  ; ALARM (9ST) PL
; rung 18
LDNOT W150.15  ; EMERG STOP:LENGTH MEASUREMENT LS FAULT
ANDNOT W159.08  ; CYCLE STOP:LENGTH MEASUREMENT FAULT CONTINUALING
ANDNOT W163.10  ; FAULT STOP:LENGTH MEASUREMENT CYCLE TIME OVER
OUT 1211.09  ; 10ST ALRAM SALL ARIA NO FAULT
; rung 19
LDNOT 1211.09  ; 10ST ALRAM SALL ARIA NO FAULT
AND P_1s
OUT W190.09  ; ALARM (10ST) PL

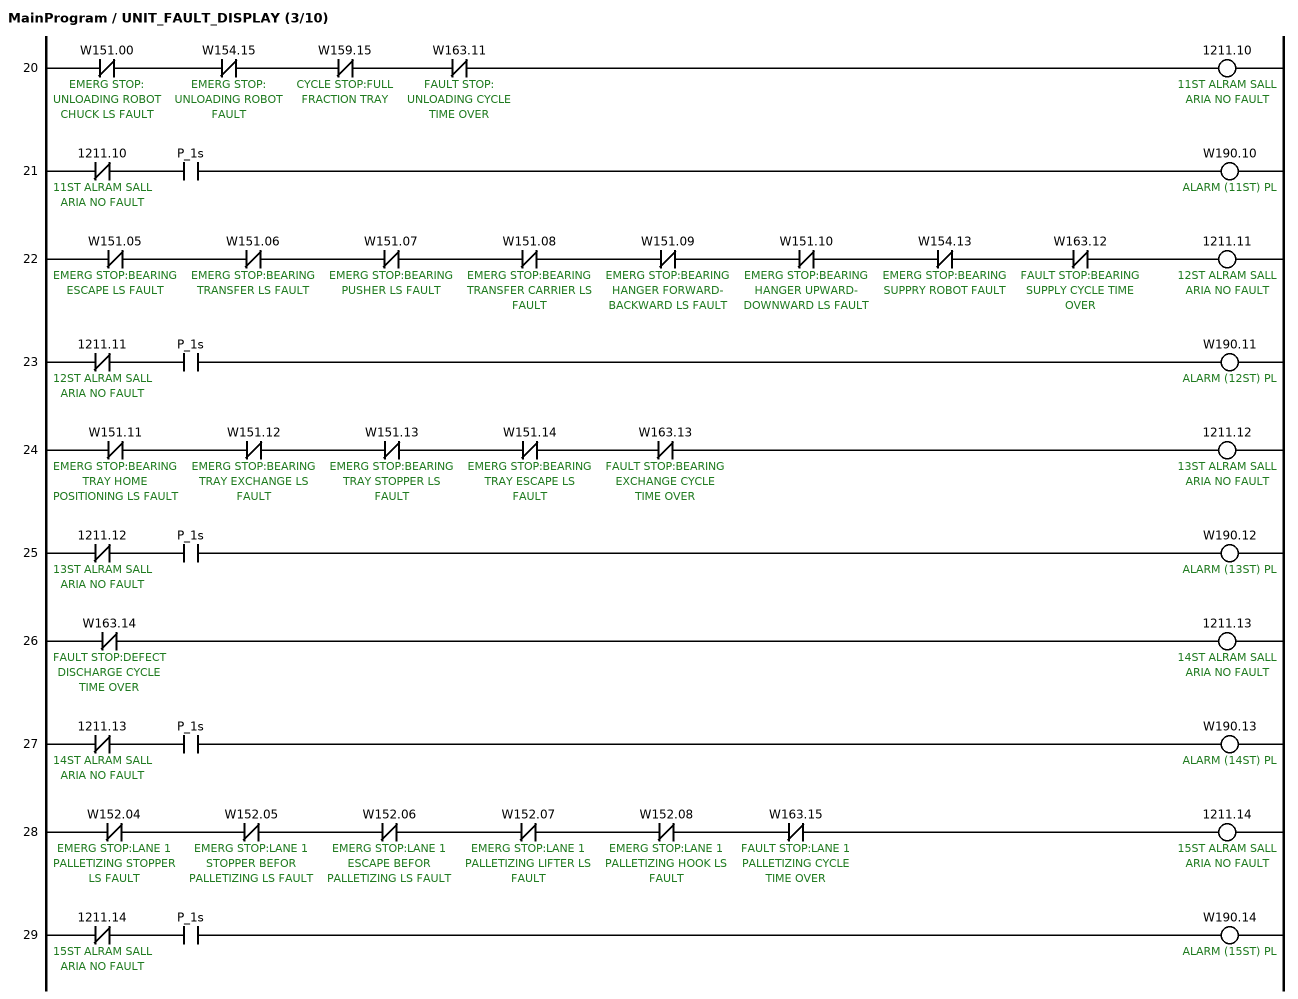
; rung 20
LDNOT W151.00  ; EMERG STOP:UNLOADING ROBOT CHUCK LS FAULT
ANDNOT W154.15  ; EMERG STOP:UNLOADING ROBOT FAULT
ANDNOT W159.15  ; CYCLE STOP:FULL FRACTION TRAY
ANDNOT W163.11  ; FAULT STOP:UNLOADING CYCLE TIME OVER
OUT 1211.10  ; 11ST ALRAM SALL ARIA NO FAULT
; rung 21
LDNOT 1211.10  ; 11ST ALRAM SALL ARIA NO FAULT
AND P_1s
OUT W190.10  ; ALARM (11ST) PL
; rung 22
LDNOT W151.05  ; EMERG STOP:BEARING ESCAPE LS FAULT
ANDNOT W151.06  ; EMERG STOP:BEARING TRANSFER LS FAULT
ANDNOT W151.07  ; EMERG STOP:BEARING PUSHER LS FAULT
ANDNOT W151.08  ; EMERG STOP:BEARING TRANSFER CARRIER LS FAULT
ANDNOT W151.09  ; EMERG STOP:BEARING HANGER FORWARD-BACKWARD LS FAULT
ANDNOT W151.10  ; EMERG STOP:BEARING HANGER UPWARD-DOWNWARD LS FAULT
ANDNOT W154.13  ; EMERG STOP:BEARING SUPPRY ROBOT FAULT
ANDNOT W163.12  ; FAULT STOP:BEARING SUPPLY CYCLE TIME OVER
OUT 1211.11  ; 12ST ALRAM SALL ARIA NO FAULT
; rung 23
LDNOT 1211.11  ; 12ST ALRAM SALL ARIA NO FAULT
AND P_1s
OUT W190.11  ; ALARM (12ST) PL
; rung 24
LDNOT W151.11  ; EMERG STOP:BEARING TRAY HOME POSITIONING LS FAULT
ANDNOT W151.12  ; EMERG STOP:BEARING TRAY EXCHANGE LS FAULT
ANDNOT W151.13  ; EMERG STOP:BEARING TRAY STOPPER LS FAULT
ANDNOT W151.14  ; EMERG STOP:BEARING TRAY ESCAPE LS FAULT
ANDNOT W163.13  ; FAULT STOP:BEARING EXCHANGE CYCLE TIME OVER
OUT 1211.12  ; 13ST ALRAM SALL ARIA NO FAULT
; rung 25
LDNOT 1211.12  ; 13ST ALRAM SALL ARIA NO FAULT
AND P_1s
OUT W190.12  ; ALARM (13ST) PL
; rung 26
LDNOT W163.14  ; FAULT STOP:DEFECT DISCHARGE CYCLE TIME OVER
OUT 1211.13  ; 14ST ALRAM SALL ARIA NO FAULT
; rung 27
LDNOT 1211.13  ; 14ST ALRAM SALL ARIA NO FAULT
AND P_1s
OUT W190.13  ; ALARM (14ST) PL
; rung 28
LDNOT W152.04  ; EMERG STOP:LANE 1 PALLETIZING STOPPER LS FAULT
ANDNOT W152.05  ; EMERG STOP:LANE 1 STOPPER BEFOR PALLETIZING LS FAULT
ANDNOT W152.06  ; EMERG STOP:LANE 1 ESCAPE BEFOR PALLETIZING LS FAULT
ANDNOT W152.07  ; EMERG STOP:LANE 1 PALLETIZING LIFTER LS FAULT
ANDNOT W152.08  ; EMERG STOP:LANE 1 PALLETIZING HOOK LS FAULT
ANDNOT W163.15  ; FAULT STOP:LANE 1 PALLETIZING CYCLE TIME OVER
OUT 1211.14  ; 15ST ALRAM SALL ARIA NO FAULT
; rung 29
LDNOT 1211.14  ; 15ST ALRAM SALL ARIA NO FAULT
AND P_1s
OUT W190.14  ; ALARM (15ST) PL

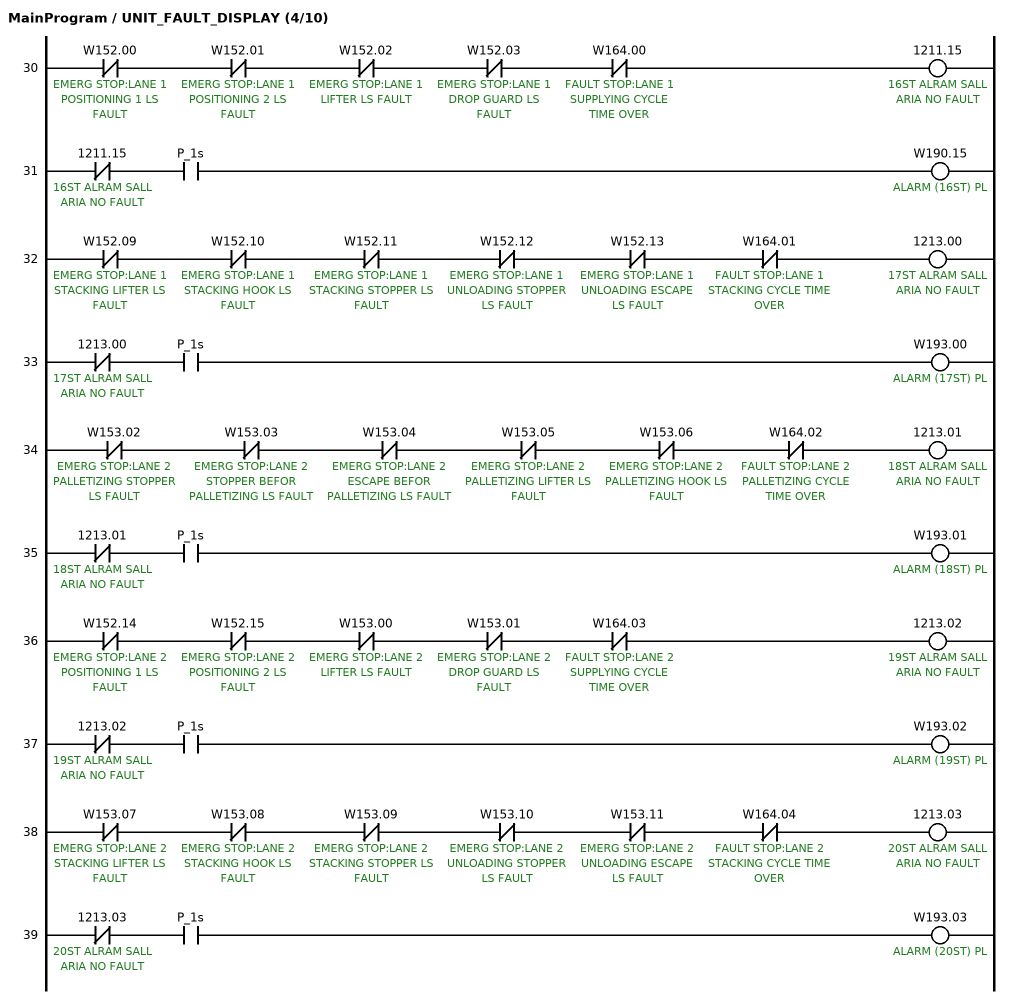
; rung 30
LDNOT W152.00  ; EMERG STOP:LANE 1 POSITIONING 1 LS FAULT
ANDNOT W152.01  ; EMERG STOP:LANE 1 POSITIONING 2 LS FAULT
ANDNOT W152.02  ; EMERG STOP:LANE 1 LIFTER LS FAULT
ANDNOT W152.03  ; EMERG STOP:LANE 1 DROP GUARD LS FAULT
ANDNOT W164.00  ; FAULT STOP:LANE 1 SUPPLYING CYCLE TIME OVER
OUT 1211.15  ; 16ST ALRAM SALL ARIA NO FAULT
; rung 31
LDNOT 1211.15  ; 16ST ALRAM SALL ARIA NO FAULT
AND P_1s
OUT W190.15  ; ALARM (16ST) PL
; rung 32
LDNOT W152.09  ; EMERG STOP:LANE 1 STACKING LIFTER LS FAULT
ANDNOT W152.10  ; EMERG STOP:LANE 1 STACKING HOOK LS FAULT
ANDNOT W152.11  ; EMERG STOP:LANE 1 STACKING STOPPER LS FAULT
ANDNOT W152.12  ; EMERG STOP:LANE 1 UNLOADING STOPPER LS FAULT
ANDNOT W152.13  ; EMERG STOP:LANE 1 UNLOADING ESCAPE LS FAULT
ANDNOT W164.01  ; FAULT STOP:LANE 1 STACKING CYCLE TIME OVER
OUT 1213.00  ; 17ST ALRAM SALL ARIA NO FAULT
; rung 33
LDNOT 1213.00  ; 17ST ALRAM SALL ARIA NO FAULT
AND P_1s
OUT W193.00  ; ALARM (17ST) PL
; rung 34
LDNOT W153.02  ; EMERG STOP:LANE 2 PALLETIZING STOPPER LS FAULT
ANDNOT W153.03  ; EMERG STOP:LANE 2 STOPPER BEFOR PALLETIZING LS FAULT
ANDNOT W153.04  ; EMERG STOP:LANE 2 ESCAPE BEFOR PALLETIZING LS FAULT
ANDNOT W153.05  ; EMERG STOP:LANE 2 PALLETIZING LIFTER LS FAULT
ANDNOT W153.06  ; EMERG STOP:LANE 2 PALLETIZING HOOK LS FAULT
ANDNOT W164.02  ; FAULT STOP:LANE 2 PALLETIZING CYCLE TIME OVER
OUT 1213.01  ; 18ST ALRAM SALL ARIA NO FAULT
; rung 35
LDNOT 1213.01  ; 18ST ALRAM SALL ARIA NO FAULT
AND P_1s
OUT W193.01  ; ALARM (18ST) PL
; rung 36
LDNOT W152.14  ; EMERG STOP:LANE 2 POSITIONING 1 LS FAULT
ANDNOT W152.15  ; EMERG STOP:LANE 2 POSITIONING 2 LS FAULT
ANDNOT W153.00  ; EMERG STOP:LANE 2 LIFTER LS FAULT
ANDNOT W153.01  ; EMERG STOP:LANE 2 DROP GUARD LS FAULT
ANDNOT W164.03  ; FAULT STOP:LANE 2 SUPPLYING CYCLE TIME OVER
OUT 1213.02  ; 19ST ALRAM SALL ARIA NO FAULT
; rung 37
LDNOT 1213.02  ; 19ST ALRAM SALL ARIA NO FAULT
AND P_1s
OUT W193.02  ; ALARM (19ST) PL
; rung 38
LDNOT W153.07  ; EMERG STOP:LANE 2 STACKING LIFTER LS FAULT
ANDNOT W153.08  ; EMERG STOP:LANE 2 STACKING HOOK LS FAULT
ANDNOT W153.09  ; EMERG STOP:LANE 2 STACKING STOPPER LS FAULT
ANDNOT W153.10  ; EMERG STOP:LANE 2 UNLOADING STOPPER LS FAULT
ANDNOT W153.11  ; EMERG STOP:LANE 2 UNLOADING ESCAPE LS FAULT
ANDNOT W164.04  ; FAULT STOP:LANE 2 STACKING CYCLE TIME OVER
OUT 1213.03  ; 20ST ALRAM SALL ARIA NO FAULT
; rung 39
LDNOT 1213.03  ; 20ST ALRAM SALL ARIA NO FAULT
AND P_1s
OUT W193.03  ; ALARM (20ST) PL

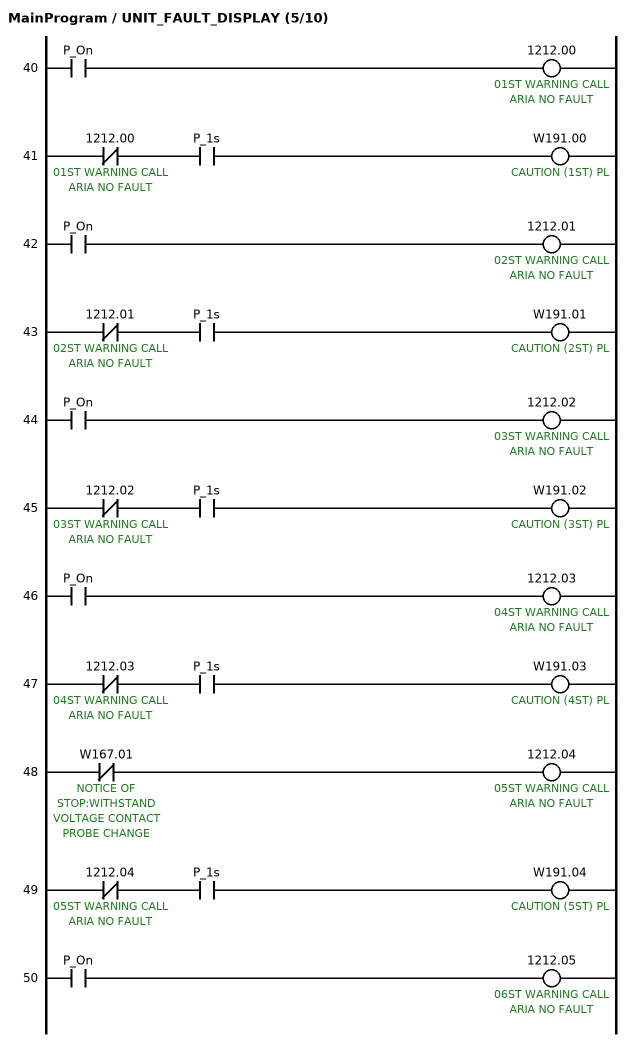
; rung 40
LD P_On
OUT 1212.00  ; 01ST WARNING CALL ARIA NO FAULT
; rung 41
LDNOT 1212.00  ; 01ST WARNING CALL ARIA NO FAULT
AND P_1s
OUT W191.00  ; CAUTION (1ST) PL
; rung 42
LD P_On
OUT 1212.01  ; 02ST WARNING CALL ARIA NO FAULT
; rung 43
LDNOT 1212.01  ; 02ST WARNING CALL ARIA NO FAULT
AND P_1s
OUT W191.01  ; CAUTION (2ST) PL
; rung 44
LD P_On
OUT 1212.02  ; 03ST WARNING CALL ARIA NO FAULT
; rung 45
LDNOT 1212.02  ; 03ST WARNING CALL ARIA NO FAULT
AND P_1s
OUT W191.02  ; CAUTION (3ST) PL
; rung 46
LD P_On
OUT 1212.03  ; 04ST WARNING CALL ARIA NO FAULT
; rung 47
LDNOT 1212.03  ; 04ST WARNING CALL ARIA NO FAULT
AND P_1s
OUT W191.03  ; CAUTION (4ST) PL
; rung 48
LDNOT W167.01  ; NOTICE OF STOP:WITHSTAND VOLTAGE CONTACT PROBE CHANGE
OUT 1212.04  ; 05ST WARNING CALL ARIA NO FAULT
; rung 49
LDNOT 1212.04  ; 05ST WARNING CALL ARIA NO FAULT
AND P_1s
OUT W191.04  ; CAUTION (5ST) PL
; rung 50
LD P_On
OUT 1212.05  ; 06ST WARNING CALL ARIA NO FAULT

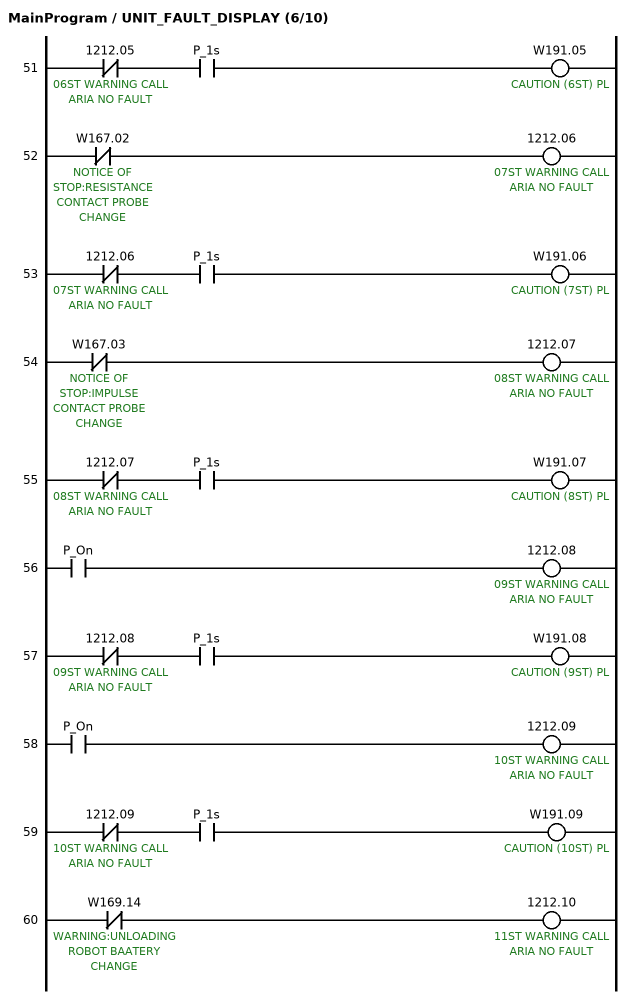
; rung 51
LDNOT 1212.05  ; 06ST WARNING CALL ARIA NO FAULT
AND P_1s
OUT W191.05  ; CAUTION (6ST) PL
; rung 52
LDNOT W167.02  ; NOTICE OF STOP:RESISTANCE CONTACT PROBE CHANGE
OUT 1212.06  ; 07ST WARNING CALL ARIA NO FAULT
; rung 53
LDNOT 1212.06  ; 07ST WARNING CALL ARIA NO FAULT
AND P_1s
OUT W191.06  ; CAUTION (7ST) PL
; rung 54
LDNOT W167.03  ; NOTICE OF STOP:IMPULSE CONTACT PROBE CHANGE
OUT 1212.07  ; 08ST WARNING CALL ARIA NO FAULT
; rung 55
LDNOT 1212.07  ; 08ST WARNING CALL ARIA NO FAULT
AND P_1s
OUT W191.07  ; CAUTION (8ST) PL
; rung 56
LD P_On
OUT 1212.08  ; 09ST WARNING CALL ARIA NO FAULT
; rung 57
LDNOT 1212.08  ; 09ST WARNING CALL ARIA NO FAULT
AND P_1s
OUT W191.08  ; CAUTION (9ST) PL
; rung 58
LD P_On
OUT 1212.09  ; 10ST WARNING CALL ARIA NO FAULT
; rung 59
LDNOT 1212.09  ; 10ST WARNING CALL ARIA NO FAULT
AND P_1s
OUT W191.09  ; CAUTION (10ST) PL
; rung 60
LDNOT W169.14  ; WARNING:UNLOADING ROBOT BAATERY CHANGE
OUT 1212.10  ; 11ST WARNING CALL ARIA NO FAULT

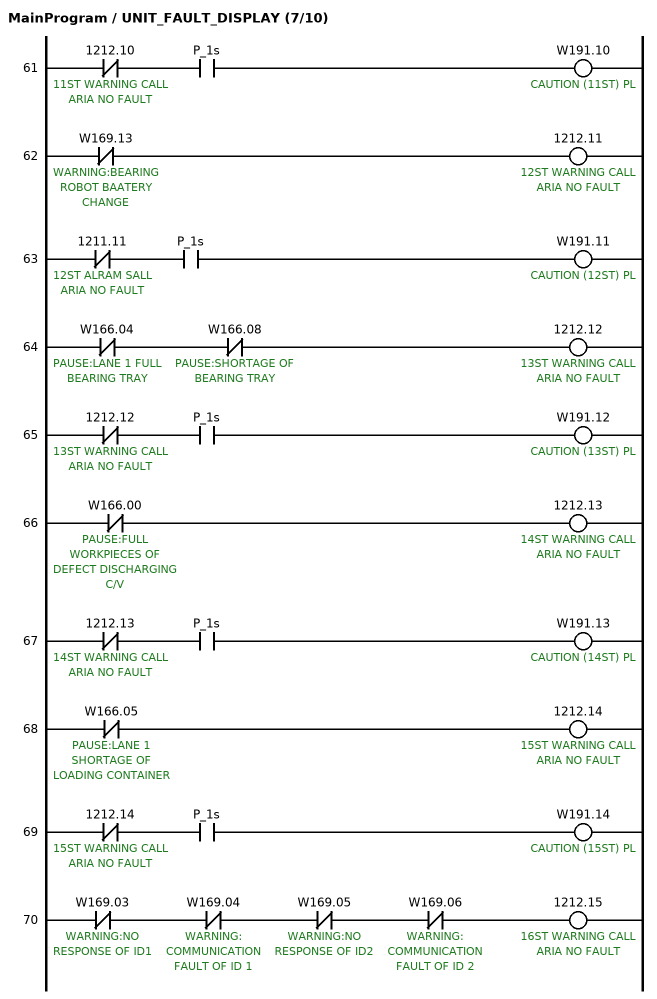
; rung 61
LDNOT 1212.10  ; 11ST WARNING CALL ARIA NO FAULT
AND P_1s
OUT W191.10  ; CAUTION (11ST) PL
; rung 62
LDNOT W169.13  ; WARNING:BEARING ROBOT BAATERY CHANGE
OUT 1212.11  ; 12ST WARNING CALL ARIA NO FAULT
; rung 63
LDNOT 1211.11  ; 12ST ALRAM SALL ARIA NO FAULT
AND P_1s
OUT W191.11  ; CAUTION (12ST) PL
; rung 64
LDNOT W166.04  ; PAUSE:LANE 1 FULL BEARING TRAY
ANDNOT W166.08  ; PAUSE:SHORTAGE OF BEARING TRAY
OUT 1212.12  ; 13ST WARNING CALL ARIA NO FAULT
; rung 65
LDNOT 1212.12  ; 13ST WARNING CALL ARIA NO FAULT
AND P_1s
OUT W191.12  ; CAUTION (13ST) PL
; rung 66
LDNOT W166.00  ; PAUSE:FULL WORKPIECES OF DEFECT DISCHARGING C/V
OUT 1212.13  ; 14ST WARNING CALL ARIA NO FAULT
; rung 67
LDNOT 1212.13  ; 14ST WARNING CALL ARIA NO FAULT
AND P_1s
OUT W191.13  ; CAUTION (14ST) PL
; rung 68
LDNOT W166.05  ; PAUSE:LANE 1 SHORTAGE OF LOADING CONTAINER
OUT 1212.14  ; 15ST WARNING CALL ARIA NO FAULT
; rung 69
LDNOT 1212.14  ; 15ST WARNING CALL ARIA NO FAULT
AND P_1s
OUT W191.14  ; CAUTION (15ST) PL
; rung 70
LDNOT W169.03  ; WARNING:NO RESPONSE OF ID1
ANDNOT W169.04  ; WARNING:COMMUNICATION FAULT OF ID 1
ANDNOT W169.05  ; WARNING:NO RESPONSE OF ID2
ANDNOT W169.06  ; WARNING:COMMUNICATION FAULT OF ID 2
OUT 1212.15  ; 16ST WARNING CALL ARIA NO FAULT

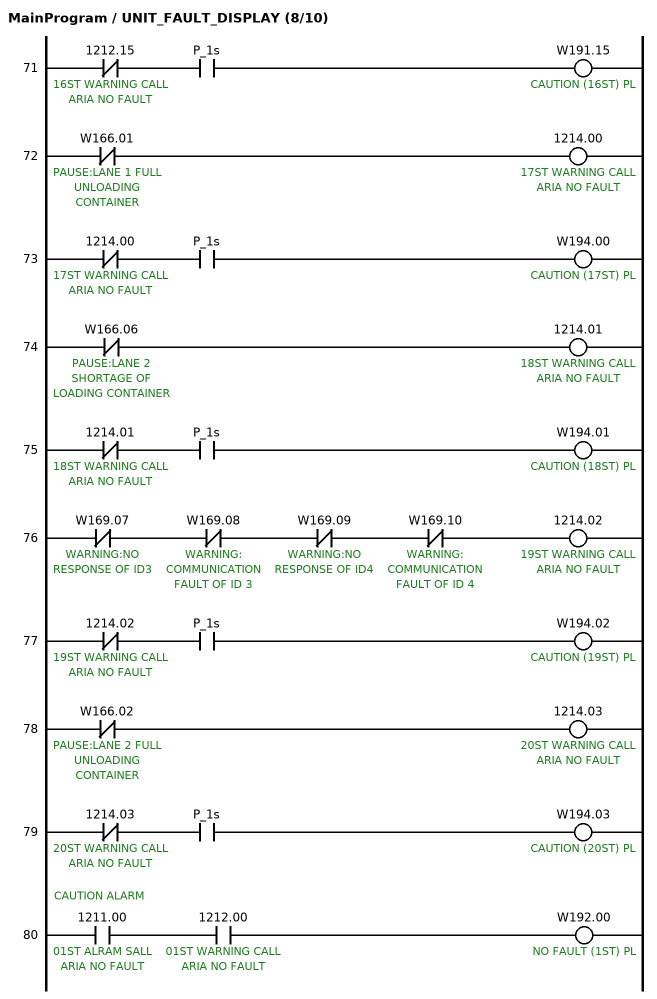
; rung 71
LDNOT 1212.15  ; 16ST WARNING CALL ARIA NO FAULT
AND P_1s
OUT W191.15  ; CAUTION (16ST) PL
; rung 72
LDNOT W166.01  ; PAUSE:LANE 1 FULL UNLOADING CONTAINER
OUT 1214.00  ; 17ST WARNING CALL ARIA NO FAULT
; rung 73
LDNOT 1214.00  ; 17ST WARNING CALL ARIA NO FAULT
AND P_1s
OUT W194.00  ; CAUTION (17ST) PL
; rung 74
LDNOT W166.06  ; PAUSE:LANE 2 SHORTAGE OF LOADING CONTAINER
OUT 1214.01  ; 18ST WARNING CALL ARIA NO FAULT
; rung 75
LDNOT 1214.01  ; 18ST WARNING CALL ARIA NO FAULT
AND P_1s
OUT W194.01  ; CAUTION (18ST) PL
; rung 76
LDNOT W169.07  ; WARNING:NO RESPONSE OF ID3
ANDNOT W169.08  ; WARNING:COMMUNICATION FAULT OF ID 3
ANDNOT W169.09  ; WARNING:NO RESPONSE OF ID4
ANDNOT W169.10  ; WARNING:COMMUNICATION FAULT OF ID 4
OUT 1214.02  ; 19ST WARNING CALL ARIA NO FAULT
; rung 77
LDNOT 1214.02  ; 19ST WARNING CALL ARIA NO FAULT
AND P_1s
OUT W194.02  ; CAUTION (19ST) PL
; rung 78
LDNOT W166.02  ; PAUSE:LANE 2 FULL UNLOADING CONTAINER
OUT 1214.03  ; 20ST WARNING CALL ARIA NO FAULT
; rung 79
LDNOT 1214.03  ; 20ST WARNING CALL ARIA NO FAULT
AND P_1s
OUT W194.03  ; CAUTION (20ST) PL
; rung 80: CAUTION ALARM
LD 1211.00  ; 01ST ALRAM SALL ARIA NO FAULT
AND 1212.00  ; 01ST WARNING CALL ARIA NO FAULT
OUT W192.00  ; NO FAULT (1ST) PL

